// Mitsubishi GX Works2 project: 231005-001- exercicios   PLC: Q03UDV

// task Task_01 (event TRUE, interval 0, priority 31): POU_01
// task Pou_St (event TRUE, interval 0, priority 31): Pou_St

PROGRAM POU_01
VAR
  x_Habilitar : BOOL;
  i_Valor01 : INT;
  i_Valor02 : INT;
  sgtOperador : STRING[32];
  Result : INT;
END_VAR
(* structured ladder/FBD written out as ST: instructions are called as NAME(EN, inputs, outputs); _pN, _eN, _tN stand for wires *)
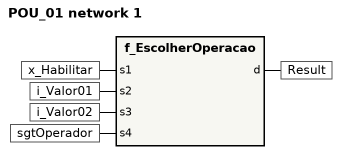
(* network 1 *)
Result := f_EscolherOperacao(x_Habilitar, i_Valor01, i_Valor02, sgtOperador);
END_PROGRAM

FUNCTION f_EscolherOperacao
VAR_INPUT
  x_Habilitar : BOOL;
  i_Valor01 : INT;
  i_Valor02 : INT;
  sgtOperador : STRING[32];
END_VAR
IF x_Habilitar THEN 
	 IF sgtOperador="+" THEN
	 	    f_EscolherOperacao:=i_Valor01+i_Valor02;
		ELSIF sgtOperador="-" THEN
			f_EscolherOperacao:=i_Valor01-i_Valor02;
		ELSIF sgtOperador="*" THEN
			f_EscolherOperacao:=i_Valor01*i_Valor02;
		ELSIF sgtOperador="/" THEN 	
			f_EscolherOperacao:=i_Valor01/i_Valor02;
		ELSIF (sgtOperador="M") OR (sgtOperador="m") THEN 
			f_EscolherOperacao:=i_Valor01 MOD i_Valor02;
		ELSE 
			f_EscolherOperacao:=32767;
		END_IF;
		
	ELSE 
	  f_EscolherOperacao:=-32767;

 END_IF;
END_FUNCTION

PROGRAM Pou_St
VAR
  resultado : ARRAY [0..9] OF INT;
END_VAR
resultado[0] := f_EscolherOperacao(TRUE , 15 , 5, "+" );
END_PROGRAM
